FUNCTION TryConvert_LWORD_TO_REAL : BOOL
VAR_INPUT
	in : LWORD;
	out : REFERENCE TO REAL;
END_VAR

out := LWORD_TO_REAL(in);
TryConvert_LWORD_TO_REAL := TRUE;

END_FUNCTION

(* stored: Version 1.1.0.1, ProductVersion 3.1.4024.12
   POU TryConvert_LWORD_TO_REAL: Id {7f8978a3-899f-4895-84d9-811abfdc7ab3}, SpecialFunc None *)
